// TwinCAT 3 PLC project main
// ProgramVersion: 3.1.4024.0
// libraries:
//   Tc2_Standard, * (Beckhoff Automation GmbH)
//   Tc2_System, * (Beckhoff Automation GmbH)
//   Tc3_Module, * (Beckhoff Automation GmbH)
// project tree:
//   / GlobalTextList.TcGTLO, PlcTask.TcTTO, Visualization Manager.TcVMO (not stored)
//   POUs/ MAIN.TcPOU
//   VISUs/ Visu.TcVIS
// real-time tasks:
//   TASK PlcTask: cycle T#10ms, priority 20, ADS port 350

CONFIGURATION main
    RESOURCE PLC ON TwinCAT3
        TASK PlcTask(INTERVAL := T#10ms, PRIORITY := 20);
        PROGRAM MAIN WITH PlcTask : MAIN;
    END_RESOURCE
END_CONFIGURATION

// ---- POUs/MAIN.TcPOU
PROGRAM MAIN
VAR
	bKnop1 : BOOL;
    bKnop2 : BOOL;
    bKnop3 : BOOL;
    bKnop4 : BOOL;
    bKnop5 : BOOL;
    bKnop6 : BOOL;
	
	bLamp : BOOL;
	outDelay: TOF;
	tijd : int;
	resetLamp: SR;
	//resetLamp: RS;
END_VAR

//In een appartementsgebouw staan in de traphal op de verschillende verdiepingen in totaal 6 drukknoppen.
//Als men één van de drukknoppen bedient gaat de verlichting branden.
//De verlichting blijft 3min. branden - tijdens de test gebruikt men 3s - vooraleer deze vanzelf uitschakelt.

//Bij iedere bediening van een drukknop zullen de lampen manueel kunnen gedoofd worden.
outDelay(IN:= bKnop1 OR bKnop2 OR bKnop3 OR bKnop4 OR bKnop5 OR bKnop6, PT:=T#10S , Q=>bLamp , ET=>);
tijd := TIME_TO_INT(outDelay.ET);
IF tijd < 10000 THEN
	if bKnop1 OR bKnop2 OR bKnop3 OR bKnop4 OR bKnop5 OR bKnop6 then
		bLamp := FALSE;
	END_IF
END_IF

END_PROGRAM

// ---- GlobalTextList.TcGTLO
TEXTLIST GlobalTextList
  533 = 'Knop 1'
  39 = 'Knop 2'
  723 = 'Knop 3'
  675 = 'Knop 4'
  283 = 'Knop 5'
  78 = 'Knop 6'
  455 = 'Label'
END_TEXTLIST

// ---- VISUs/Visu.TcVIS
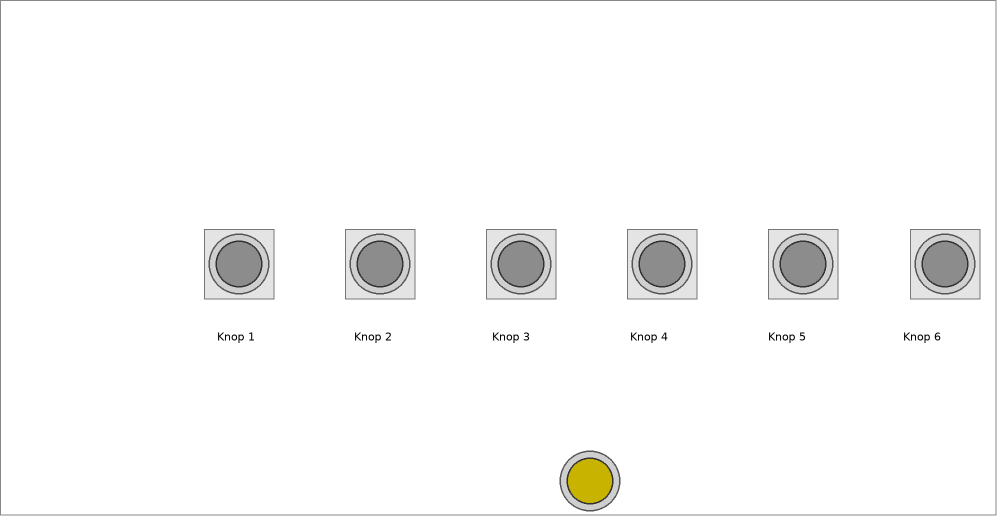
VISUALIZATION Visu  // 997x516
    PushSwitch (486,229 70x70), variable: MAIN.bKnop3, behaviour: TAP, style: Switch-PushSwitch-Gray
    PushSwitch (204,229 70x70), variable: MAIN.bKnop1, behaviour: TAP, style: Switch-PushSwitch-Gray
    PushSwitch (345,229 70x70), variable: MAIN.bKnop2, behaviour: TAP, style: Switch-PushSwitch-Gray
    PushSwitch (627,229 70x70), variable: MAIN.bKnop4, behaviour: TAP, style: Switch-PushSwitch-Gray
    PushSwitch (768,229 70x70), variable: MAIN.bKnop5, behaviour: TAP, style: Switch-PushSwitch-Gray
    PushSwitch (910,229 70x70), variable: MAIN.bKnop6, behaviour: TAP, style: Switch-PushSwitch-Gray
    Label (161,322 150x30), "Knop 1"
    Label (298,322 150x30), "Knop 2"
    Label (436,322 150x30), "Knop 3"
    Label (574,322 150x30), "Knop 4"
    Label (712,322 150x30), "Knop 5"
    Label (847,322 150x30), "Knop 6"
    Lamp1 (555,446 70x70), variable: MAIN.bLamp, style: Lamp-Lamp1-Yellow
END_VISUALIZATION
